// TwinCAT 3 PLC project motor_test
// ProgramVersion: 3.1.0.8
// libraries:
//   VisuElem3DPath, 3.5.4.0 (System)
//   VisuElemMeter, 3.5.4.0 (System)
//   VisuElems, 3.5.4.10 (System)
//   VisuElemsSpecialControls, 3.5.4.10 (System)
//   VisuElemsWinControls, 3.5.4.10 (System)
//   VisuElemTextEditor, 3.5.4.0 (System)
//   visuinputs, 3.5.4.0 (system)
//   VisuNativeControl, 3.5.4.0 (System)
//   Tc2_Standard, * (Beckhoff Automation GmbH)
//   Tc2_System, * (Beckhoff Automation GmbH)
//   Tc3_Interfaces, * (Beckhoff Automation GmbH)
//   Tc3_Module, * (Beckhoff Automation GmbH)
//   Tc2_MC2,3.3.8.0,Beckhoff Automation GmbH
//   Tc2_SerialCom,3.3.3.0,Beckhoff Automation GmbH
// project tree:
//   / GlobalTextList.TcGTLO, PlcTask.TcTTO
//   POUs/ MAIN.TcPOU

CONFIGURATION motor_test
    RESOURCE PLC ON TwinCAT3
        TASK PlcTask(INTERVAL := T#10ms, PRIORITY := 20);
        PROGRAM MAIN WITH PlcTask : MAIN;
    END_RESOURCE
END_CONFIGURATION

// ---- POUs/MAIN.TcPOU
PROGRAM MAIN
VAR
	axisX, axisY : AXIS_REF;
	diX, diY AT %I* : BOOL;
	bEnable : BOOL;
	powerX, powerY : MC_Power;
	resetX, resetY : MC_Reset;
	homeX, homeY : MC_Home;
	moveAbsY, moveAbsY : MC_MoveAbsolute;
END_VAR

END_PROGRAM
